// TIA Portal V20 export
TYPE "typeCmControlNode"
// stored: Namespace Unit1.Em1
   STRUCT
      interlock : "Unit1.Em1.typeCmControlNodeInterlock";
   END_STRUCT;
END_TYPE
